//----------------------------------------------------------------------------//
//            Copyright 2018 Rieckermann Engineering Operations               //
//                Automatically Generated File - Do Not Edit                  //
//----------------------------------------------------------------------------//
// Class:       ifbDI1                                                        //
// Description: Instances of DI1                                              //
//                                                                            //
// General alarm single digital input.                                        //
//----------------------------------------------------------------------------//
// Revision history:                                                          //
// Rev By               Date        CC        Note                            //
// 2.0 David Paspa      05-Jan-2018 NA        Reboot for S7-1500.             //
// 0.6 Khairul Basar    12-Oct-2009 CC-09/016 IN_REQ_MODE is assigned to      //
//                                            Toggle.                         //
// 0.5 Khairul Basar    03-Oct-2009 CC-09/016 PSH_parameters corrected.       //
// 0.4 Khairul Basar    15-Sep-2009 CC-09/016 PSA_1010 DI_USER assigned       //
//                                            correctly.                      //
// 0.3 Khairul Basar    09-Sep-2009 CC-09/016 I/O assignment associated with  //
//                                            corresponding Instance is       //
//                                            corrected.                      //
// 0.2 Khairul Basar    31-Aug-2009 CC-09/016 Mode=1 initialized.             //
//                                            Instance comment added.         //
// 0.1 Khairul Basar    03-Aug-2009 NA        Initial design.                 //
//----------------------------------------------------------------------------//
FUNCTION_BLOCK "ifbDI1"
TITLE = Instances of DI1 General alarm single digital input Normally ON
{ S7_Optimized_Access := 'TRUE' }
AUTHOR : REO
NAME : ifbDI1
VERSION : 2.0

//----------------------------------------------------------------------------//
// Declare the instance objects of the class:                                 //
//----------------------------------------------------------------------------//
VAR
@@TEMPLATE_BEGIN@@
    @@INSTANCE@@ : "fbDI1";  // @@DESCRIPTION@@
@@TEMPLATE_END@@
END_VAR

BEGIN
@@TEMPLATE_BEGIN|createInstances@@
NETWORK
TITLE = @@INSTANCE@@ : Unique ID
    //------------------------------------------------------------------------//
    // Set the instance unique ID:                                            //
    //------------------------------------------------------------------------//
    L "dbCONST".BLK.ID.@@INSTANCE@@;
    T #@@INSTANCE@@.mc.ME;

NETWORK
TITLE = @@INSTANCE@@ : Owner
    //------------------------------------------------------------------------//
    // Set the instance owner:                                                //
    //------------------------------------------------------------------------//
    L "dbCONST".BLK.ID.@@PARENT@@;
    T #@@INSTANCE@@.mc.OWNER;

NETWORK
TITLE = @@INSTANCE@@ : Safe Command on restart
    //------------------------------------------------------------------------//
    // Set the safe command if restarting the PLC:                            //
    //------------------------------------------------------------------------//
    A "flagFirstScanRestart";
    JCN _notRestart_@@COUNTER|1@@;
    L "dbCONST".BLK.DI1.SAFE.CMD;
    T #@@INSTANCE@@.mc.CMD_SAFE;
_notRestart_@@COUNTER@@:   NOP 0;

NETWORK
TITLE = @@INSTANCE@@ : @@DESCRIPTION@@
    //------------------------------------------------------------------------//
    // Call the class function to process the instance:                       //
    //------------------------------------------------------------------------//
    CALL #@@INSTANCE@@
    (   DI_Auto              := "@@INSTANCE@@-DI"
    );

@@TEMPLATE_END@@
END_FUNCTION_BLOCK
